{attribute addProperty BoxType "AX8206-0000-0041-0041"}
{attribute addProperty Id "Ch_B_Following_error_actual_valueAT %I*DINT324"}
{attribute addProperty CRC "1639779927"}
{attribute addProperty SizeInBites "32"}
{attribute addProperty SizeInBytes "4"}
TYPE Ch_B_PositionControl_Inputs_61BD0E57 :
STRUCT
	{attribute addProperty Name "Ch_B_Following_error_actual_value"}
	Ch_B_Following_error_actual_value AT %I* : DINT;
END_STRUCT
END_TYPE

(* stored: Version 1.2.0.0, ProductVersion 3.1.4024.9
   DUT Ch_B_PositionControl_Inputs_61BD0E57: Id {053fcf56-e0e0-4e81-8c32-d094509b2098} *)
